PROGRAM MAIN
VAR
	sVersion: STRING:='1.0.0';
	M1:FB_DriveVirtual;
	M1Link:FB_NcAxis;
	bLimitFwd AT %I*: BOOL;
	bLimitBwd AT %I*: BOOL;
	bHomeSensor AT %I*: BOOL;
	bOutput1 AT %Q*: BOOL:= TRUE;
	bOutput2 AT %Q*: BOOL:= TRUE;
	bOutput3 AT %Q*: BOOL:= TRUE;
	bOutput4 AT %Q*: BOOL:= TRUE;
	bOutput5 AT %Q*: BOOL:= TRUE;
	bOutput6 AT %Q*: BOOL:= TRUE;
	bOutput7 AT %Q*: BOOL:= TRUE;
	bOutput8 AT %Q*: BOOL:= TRUE;
END_VAR

act();

ACTION ACT:
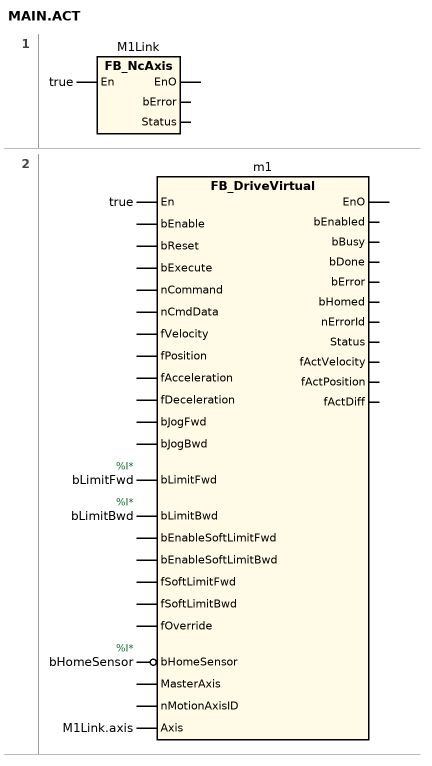
// NETWORK 1
M1Link(En := true); // FB_NcAxis

// NETWORK 2
//   bLimitFwd: AT %I*
//   bLimitBwd: AT %I*
//   bHomeSensor: AT %I*
m1(
    En := true,
    bLimitFwd := bLimitFwd,
    bLimitBwd := bLimitBwd,
    bHomeSensor := NOT bHomeSensor,
    Axis := M1Link.axis); // FB_DriveVirtual
END_ACTION

END_PROGRAM

(* stored: Version 1.1.0.1, ProductVersion 3.1.0.36
   POU MAIN: Id {68d5c4cd-ed5a-46ef-a7cd-a34a6aaecb11}, SpecialFunc None
   Action ACT: Id {d90d5e50-7562-49a7-958d-fc203dcb8912} *)
